// TIA Portal V16 export
// export: Created 2020-03-17T19:26:44.1402669Z, ExportSetting None, DisplayName Totally Integrated Automation Portal, DisplayVersion V16, DisplayName TIA Portal Version Control Interface, DisplayVersion V16, DisplayName TIA Portal Openness, DisplayVersion V16, DisplayName STEP 7 Professional, DisplayVersion V16, DisplayName STEP 7 Safety, DisplayVersion V16, DisplayName WinCC Advanced, DisplayVersion V16
DATA_BLOCK "StepData"   // DB1
{ S7_Optimized_Access := 'TRUE' }
// stored: MemoryReserve 100
   VAR RETAIN
      Steps : Array[0..99] of "Step";
   END_VAR
   VAR
      Values : "StepValues";
   END_VAR
BEGIN
END_DATA_BLOCK
